{attribute 'qualified_only'}
VAR_GLOBAL
	// In-Vacuum Motion
    {attribute 'pytmc':='pv: DREAM:DGPD:MMT:X'}
    {attribute 'TcLinkTo' := '
        .nRawEncoderDINT        :=TIID^Device 1 (EtherCAT)^TMO-DREAM-SMARACT-03^DREAM:DGPD:MMT:X^mode/status/pos/fError TxPDO^Position Actual Value;
    '}
    M9 : ST_MotionStage:= (
            sName:='DREAM:DGPD:MMT:X'
    );

    {attribute 'pytmc':='pv: DREAM:DGPD:MMT:Y'}
    {attribute 'TcLinkTo' := '
        .nRawEncoderDINT        :=TIID^Device 1 (EtherCAT)^TMO-DREAM-SMARACT-03^DREAM:DGPD:MMT:Y^mode/status/pos/fError TxPDO^Position Actual Value;
    '}
    M10 : ST_MotionStage:= (
		sName:='DREAM:DGPD:MMT:Y'
    );

    {attribute 'pytmc':='pv: DREAM:DGPD:MMT:Z'}
//     {attribute 'TcLinkTo' := '
//      .nRawEncoderDINT        :=TIID^Device 1 (EtherCAT)^TMO-DREAM-SMARACT-03^DREAM:DGPD:MMT:Z^mode/status/pos/fError TxPDO^Position Actual Value;
//     '}
    M11 : ST_MotionStage:= (
                sName:='DREAM:DGPD:MMT:Z'
    );

    {attribute 'pytmc':='pv: DREAM:DGPD:MMT:RET'}
    {attribute 'TcLinkTo' := '
        .nRawEncoderDINT        :=TIID^Device 1 (EtherCAT)^TMO-DREAM-SMARACT-03^DREAM:DGPD:MMT:RET^mode/status/pos/fError TxPDO^Position Actual Value;
    '}
    M12 : ST_MotionStage:= (
        sName:='DREAM:DGPD:MMT:RET'
    );

END_VAR

(* stored: Version 1.1.0.1
   GVL Main_Sim: Id {7eb6578c-9995-479d-b58a-4f9eafc09fc0} *)
